{attribute 'qualified_only'}
{attribute 'strict'}
TYPE EFeedbackMsgEol :
(
	IdMsg := 10,
    CustomMsg
);
END_TYPE

(* stored: Version 1.1.0.1, ProductVersion 3.1.4024.4
   DUT EFeedbackMsgEol: Id {85f9f954-adcb-4ae8-a1dd-22776bb5a8f9} *)
